// TIA Portal V19 export
FUNCTION "Prod_TODO_FindIndex_Of_FirstExecutable" : Int   // FC76, LAD
TITLE = TROVA L'INDICE SU ARRAY TODO CHE CONTIENE IL PRIMO ORDINE ESEGUIBILE
// stored: SetENOAutomatically false
   VAR_TEMP
      i : Int;
      RETVAL : DInt;
   END_VAR
BEGIN

REGION Network 1 (SCL): Ricerca ordine eseguibile = Con dati corretti e che usa lo stesso profilo del SETUP o del Profilo in lavoro
   #Prod_TODO_FindIndex_Of_FirstExecutable := 0;


   // Pulisci i gap
   // 

   FOR #i := 1 TO "PROD_TODO_ITEMS" DO

       #RETVAL := "PROD_item_Clear_GAP"("Production".O_TODO);

       IF #RETVAL <> "PROD_FUN_RESULT_CLEAR_GAP_DONE" THEN
           EXIT;
       END_IF;


   END_FOR;








   // Ricerca su O_TODO la prima posizione con ordine eseguibile
   // 
   FOR #i := 1 TO "PROD_TODO_ITEMS" DO

       #RETVAL := "Prod_Item_Check_CanGoinProduction"("Production".O_TODO[#i]);

       IF #RETVAL >= 0 THEN
           #Prod_TODO_FindIndex_Of_FirstExecutable := #i;
           EXIT;
       END_IF;

   END_FOR;
END_REGION

REGION Network 2: +
END_REGION

REGION Network 3: +
END_REGION

REGION Network 4: +
END_REGION
END_FUNCTION
